TYPE ST_Datalog_event :
STRUCT
	s_header		: STRING;
	s_data			: STRING;			
END_STRUCT
END_TYPE

(* stored: Version 1.1.0.1, ProductVersion 3.1.4024.12
   DUT ST_Datalog_event: Id {cf6b50f2-103e-460d-b181-741086fde1a6} *)
